Staubli VAL3: start.pgx

program start()
begin
  call MotionPage()
end
